TYPE ST_System_DLK_Stellwert :
STRUCT
	Anford_Stellventil		: BOOL;
	Anford_Pumpe			: BOOL;
	Anford_Kompressor		: BOOL;
	Einschaltperiode_Max	: TIME := T#5S;
	Einschalten				: BOOL;
END_STRUCT
END_TYPE

(* stored: Version 1.1.0.1, ProductVersion 3.1.4024.9
   DUT ST_System_DLK_Stellwert: Id {128a1438-9815-4447-9290-feb09e685178} *)
